FUNCTION_BLOCK PUBLIC StringBuilder IMPLEMENTS  IStringBuilder, ILimitedStringBuilder
VAR
	{attribute 'hide'}
	_workString:STRING;
END_VAR

METHOD PUBLIC Append : IStringBuilder // Append text to t current build string.
VAR_INPUT
	text:STRING; //Text to append to current build string
END_VAR
_workString:= Concat(_workString,text);
Append := THIS^;
END_METHOD

METHOD PUBLIC InsertAtLocation : IStringBuilder
VAR_INPUT
	Text:STRING;
	Position:INT;
END_VAR
_workString := Tc2_Standard.INSERT(_WorkSTring,Text,Position);
InsertAtLocation  := THIS^;
END_METHOD

METHOD PUBLIC Reset : ILimitedStringBuilder //Reset current build string to an empty string.
_workString:='';
Reset := THIS^;
END_METHOD

METHOD PUBLIC ToString : STRING //Returns current build string.
ToString := _workString;
END_METHOD

END_FUNCTION_BLOCK

(* stored: Version 1.1.0.1, ProductVersion 3.1.4024.0
   POU StringBuilder: Id {368e5049-935b-4562-a874-cb9be5225f7d}, SpecialFunc None
   Method Append: Id {3f45997e-6006-457f-9a9a-30ac281e8f8a}
   Method InsertAtLocation: Id {b2ed9ced-aca1-4991-af8e-c808997da606}
   Method Reset: Id {f04f2676-7659-44a8-87c7-48fdd5328c04}
   Method ToString: Id {8c20dc6d-f3fa-4203-b887-d1b9b96ecacc} *)
